FUNCTION_BLOCK INTERNAL FB_PwmLightTowerComponent IMPLEMENTS I_PwmLightTowerComponent, I_LightTowerComponent
VAR_INPUT
END_VAR
VAR_OUTPUT
END_VAR
VAR
	_active		: BOOL;
	_interval	: TIME;
	_state		: BOOL;
	fbPulseGenerator	: ZigaLibs_Core.FB_PulseGenerator( tPeriod := _interval, fDutyCycle := 50);
END_VAR

fbPulseGenerator.Enable := TRUE;
_state := NOT fbPulseGenerator.Execute() AND _active;

METHOD Activate
_active := TRUE;
END_METHOD

METHOD Deactivate
_active := FALSE;
END_METHOD

METHOD SetInterval : I_LightTowerComponent
VAR_INPUT
	tInterval : TIME;
END_VAR
_interval := tInterval;
SetInterval := THIS^;
END_METHOD

PROPERTY State : BOOL
GET
State := _state;
END_GET
END_PROPERTY

END_FUNCTION_BLOCK

(* stored: Version 1.1.0.1, ProductVersion 3.1.4024.13
   POU FB_PwmLightTowerComponent: Id {5c19a601-f767-0344-0722-2f67269d801d}, SpecialFunc None
   Method Activate: Id {e3b6b1e8-08ce-0fda-3e26-386c2ccd280f}
   Method Deactivate: Id {021e6582-c51a-0979-24d7-fe7c84929d70}
   Method SetInterval: Id {49bc24d2-ba9f-0516-1ca8-4c245f14c997}
   Property State: Id {1e26d076-f5b2-03ad-1322-885e2d036ceb}
   Get Get: Id {fef036ac-abc9-08cc-30e8-2c08089e919d} *)
